{attribute 'qualified_only'}
VAR_GLOBAL
	Alt				: Axis_Ref := Alt;
	Az				: Axis_Ref := Az;
END_VAR

(* stored: Version 1.1.0.1
   GVL GVL: Id {77dabe38-abf3-4946-9c1f-21aeb2ae5804} *)
